FUNCTION_BLOCK PUBLIC FB_FactoryIO_ModbusTCP
VAR_INPUT
	sIPAddr : STRING[15]:='127.0.0.1'; // '127.0.0.1'
	nTCPPort : UINT:=505; // 505
	nUnitID : BYTE:=255; // 255
	
	// **** Configuration des array en fonction de la configuration FactoryIO
	OutputReg : ARRAY [0..7] OF INT;
	// Outpus traités
	bOutput1 : ARRAY [0..15] OF BOOL;
	bOutput2 : ARRAY [0..15] OF BOOL;
	
END_VAR

VAR_OUTPUT
	bBusy: BOOL;
	bError: BOOL;
	// *** Configuration des array en fonction de la configuration FactoryIO
	InputReg : ARRAY [0..7] OF INT; // ex. input register 8 [0..7] pour les mesures analogiques
	// Inputs traités
	bInput1 : ARRAY [0..15] OF BOOL;
	bInput2 : ARRAY [0..15] OF BOOL;
	
END_VAR
	
VAR
	// Instances
	fb_MBReadInputs : FB_MBReadInputs; // Instance de la fonction FB_MBReadInputs de la lib Tc2_ModbusSrv
	fb_MBReadInputRegs : FB_MBReadInputRegs;
	fb_MBWriteCoils : FB_MBWriteCoils;
	fb_MBWriteRegs : FB_MBWriteRegs ;
	
	fb_Word_To_Bool : FB_Word_To_Bool; // Instance commune
	fb_Bool_To_Word: FB_Bool_To_Word ; // Instance commune
	
	// *** Configuration des array en fonction de la configuration FactoryIO
	Input : ARRAY [0..1] OF WORD; // ex. input digital 16 [0..0] /  input digital 32 [0..1]
	// **** Configuration des array en fonction de la configuration FactoryIO
	Output : ARRAY [0..1] OF WORD;
	
	// Busy Error interne à la fonciton
	bBusyInput: ARRAY [1..4] OF BOOL;
	bErrorInput: ARRAY [1..4] OF BOOL;

END_VAR


// Traitement des bool représentant les inputs
fb_Word_To_Bool(inWord := Input[0],
				outArrayOfBool => bInput1);
fb_Word_To_Bool(inWord := Input[1],
				outArrayOfBool => bInput2);
				
// Traitement des bool représentant les outputs
fb_Bool_To_Word(inArrayOfBool := bOutput1,
				outWord => Output[0]);
fb_Bool_To_Word(inArrayOfBool := bOutput2,
				outWord => Output[1]);	
				

// Busy si au moins 1 busy
IF bBusyInput[1] OR bBusyInput[2] OR bBusyInput[3] OR bBusyInput[4] THEN
	bBusy := 1;
ELSE
	bBusy := 0;
END_IF

// Error si au moins 1 busy
IF bErrorInput[1] OR bErrorInput[2] OR bErrorInput[3] OR bErrorInput[4] THEN
	bError := 1;
ELSE
	bError := 0;
END_IF

METHOD PUBLIC Read_Input
fb_MBReadInputs(
	sIPAddr := sIPAddr,
	nTCPPort := nTCPPort,
	nUnitID := nUnitID,
	nQuantity := SIZEOF(Input)*8, // Nombre de bits à lire SIZEOF(nb byte * bits dans 1 byte)
	nMBAddr := 0,
	cbLength := SIZEOF(Input),
	pDestAddr := ADR(Input),
	bExecute := TRUE,
	tTimeout := T#1S,
	bBusy => bBusyInput[1],
	bError => bErrorInput[1],
	nErrId => ,
	cbRead => ,
 );
fb_MBReadInputs(bExecute := FALSE);
END_METHOD

METHOD PUBLIC Read_InputRegister
fb_MBReadInputRegs(
	sIPAddr := sIPAddr,
	nTCPPort := nTCPPort,
	nUnitID := nUnitID,
	nQuantity := SIZEOF(InputReg)/2,
	nMBAddr := 0,
	cbLength := SIZEOF(InputReg),
	pDestAddr := ADR(InputReg),
	bExecute := TRUE,
	tTimeout := T#1S,
	bBusy => bBusyInput[2],
	bError => bErrorInput[2],
	nErrId => ,
	cbRead => ,
 );
fb_MBReadInputRegs(bExecute := FALSE);
END_METHOD

METHOD PUBLIC Write_Output
fb_MBWriteCoils(
	sIPAddr := sIPAddr,
	nTCPPort := nTCPPort,
	nUnitID := nUnitID,
	nQuantity := SIZEOF(Output)*8,
	nMBAddr := 0,
	cbLength := SIZEOF(Output),
	pSrcAddr := ADR(Output),
	bExecute := TRUE,
	tTimeout := T#1S,
	bBusy => bBusyInput[3],
	bError => bErrorInput[3],
	nErrId => ,
 );
fb_MBWriteCoils(bExecute := FALSE);
END_METHOD

METHOD PUBLIC Write_OutputRegister
fb_MBWriteRegs(
	sIPAddr := sIPAddr,
	nTCPPort := nTCPPort,
	nUnitID := nUnitID,
	nQuantity := SIZEOF(OutputReg)/2,
	nMBAddr := 0,
	cbLength := SIZEOF(OutputReg),
	pSrcAddr := ADR(InputReg),
	bExecute := TRUE,
	tTimeout := T#1S,
	bBusy => bBusyInput[4],
	bError => bErrorInput[4],
	nErrId => ,
 );
fb_MBWriteRegs(bExecute := FALSE);
END_METHOD

END_FUNCTION_BLOCK

(* stored: Version 1.1.0.1, ProductVersion 3.1.4024.11
   POU FB_FactoryIO_ModbusTCP: Id {ef99659b-bb0e-494d-8cf7-6072e7c46a5c}, SpecialFunc None
   Method Read_Input: Id {114b7d6d-1641-41a1-9a37-c80540c5b291}
   Method Read_InputRegister: Id {49627f2a-4539-4976-b388-686bcf311a5b}
   Method Write_Output: Id {434578e9-d9ba-4b29-902c-1d1c5a578d51}
   Method Write_OutputRegister: Id {7e2de503-8972-44d8-bb85-cbb1ce981c07} *)
